{attribute 'call_after_init'}
FUNCTION_BLOCK FB_Printer_Test EXTENDS TcUnit.FB_TestSuite IMPLEMENTS TcUnit.I_RunnableTestSuite
VAR
    Assert : TcUnit.FB_Assert;
    
    getFailureMessageString_Printer: UnitTestPrinter;
    getFailureMessageINT_Printer: UnitTestPrinter;
END_VAR

METHOD FB_init : BOOL
VAR_INPUT
	bInitRetains : BOOL; // if TRUE, the retain variables are initialized (warm start / cold start)
	bInCopyCode : BOOL;  // if TRUE, the instance afterwards gets moved into the copy code (online change)
END_VAR
SUPER^.RegisterTestSuite(THIS^);
END_METHOD

METHOD RunTests : TCUNIT.E_TestSuiteRunState
Test_GetFailureMessageString();
Test_GetFailureMessageINT();

RunTests := TCUNIT.E_TestSuiteRunState.FINISHED;
END_METHOD

METHOD Test_GetFailureMessageINT
VAR
    expected: MaxString;
    actual: MaxString;
    
    expectedTestValue: INT;
    actualTestValue: INT;
    message: MaxString;
    path: MaxString;
END_VAR
TEST('Test_GetFailureMessageINT');

expected := 'FAILED TEST $'FB_TestSuite_Test$', EXP: 1234, ACT: 1235, MSG: INTs do not match';

expectedTestValue := 1234;
actualTestValue := 1235;
message := 'INTs do not match';
path := 'FB_TestSuite_Test';
actual := getFailureMessageINT_Printer.getFailureMessage(expectedTestValue, actualTestValue, message, path);

Assert.AssertEquals_STRING(expected, actual, 'Get Failure Message INT does not match');
END_METHOD

METHOD Test_GetFailureMessageString
VAR
    expected: MaxString;
    actual: MaxString;
    
    expectedTestValue: MaxString;
    actualTestValue: MaxString;
    message: MaxString;
    path: MaxString;
END_VAR
TEST('Test_GetFailureMessageString');

expected := 'FAILED TEST $'FB_TestSuite_Test$', EXP: hello, ACT: world, MSG: Strings do not match';

expectedTestValue := 'hello';
actualTestValue := 'world';
message := 'Strings do not match';
path := 'FB_TestSuite_Test';
actual := getFailureMessageString_Printer.getFailureMessage(expectedTestValue, actualTestValue, message, path);

Assert.AssertEquals_STRING(expected, actual, 'Get Failure Message String does not match');
END_METHOD

END_FUNCTION_BLOCK

(* stored: Version 1.1.0.1, ProductVersion 3.1.4022.12
   POU FB_Printer_Test: Id {3959c355-b6db-4f36-95b0-00d7b37d0885}, SpecialFunc None
   Method FB_init: Id {071a2ba1-435a-4be7-a90e-47ffadbf0dea}
   Method RunTests: Id {7d1a596a-5eb5-45d5-8c83-5cfb1d76d03e}
   Method Test_GetFailureMessageINT: Id {da0e0c8f-411c-4f45-a2bf-486555123498}
   Method Test_GetFailureMessageString: Id {d460dccf-336c-4386-a8ef-ee0120ae7e7f} *)
